FUNCTION_BLOCK FB_distSensor2011
VAR
	nSensor AT %I* 	: INT;
	fHeightVal 		: REAL;
	fSensorAvg		: REAL;
	nAvgSensorCount : INT;
	fPrevHeight		: REAL;
	fLowBound 		: REAL := 257; // mm's at 4 mA on sensor
	fHighBound		: REAL := 1226; // mm's at 20 mA on sensor
END_VAR

PROPERTY height : REAL //Distance in inches
GET
//height := (((INT_TO_REAL(sensor)/32767)*3000)+50)/25.4;
IF nAvgSensorCount <= 25 THEN
	nAvgSensorCount := nAvgSensorCount + 1;
	fSensorAvg := fSensorAvg + ((INT_TO_REAL(nSensor))/25);
	fHeightVal := fPrevHeight;
	height := fPrevHeight;
ELSE 
	height := (((fSensorAvg/43519)*fHighBound)+fLowBound)/25.4;
	fPrevHeight := height;
	fSensorAvg := 0;
	nAvgSensorCount := 0;
	fHeightVal := height;
END_IF
END_GET
END_PROPERTY

END_FUNCTION_BLOCK

(* stored: Version 1.1.0.1, ProductVersion 3.1.4024.13
   POU FB_distSensor2011: Id {e6af5067-769c-4f54-8a1a-703851786096}, SpecialFunc None
   Property height: Id {55486666-a5d0-4146-a773-54d9595d890a}
   Get Get: Id {83f0b03b-06ce-40a7-81d3-c2a3c68c7185} *)
